FUNCTION "LAnyAxis_UnpubHaltPosAxis" : Void
{ S7_Optimized_Access := 'TRUE' }
AUTHOR : 'tech.team.motioncontrol@siemens.com'
FAMILY : AnyAxis
VERSION : 1.0
   VAR_INPUT
      axis {InstructionName := 'TO_PositioningAxis'; LibVersion := '6.0'} : TO_PositioningAxis;
   END_VAR

   VAR_IN_OUT
      instMC {InstructionName := 'MC_HALT'; LibVersion := '6.0'} : MC_HALT;
   END_VAR


BEGIN
	// Call of MC_Instruction
	#instMC(Axis := #axis);
END_FUNCTION

